FUNCTION_BLOCK ResetModulesVisitor IMPLEMENTS I_ModuleVisitor, I_TaskResult
VAR
	{attribute 'hide'}
	Resettable : I_Resettable;
	{attribute 'hide'}
	Result : I_TaskResult;
	{attribute 'hide'}
	_Busy : BOOL;
	{attribute 'hide'}
	_Error : BOOL;
	{attribute 'hide'}
	_ErrorId	: UDINT;
	ErrorModule : I_Module;
END_VAR

{attribute 'monitoring' := 'call'}
PROPERTY Busy : BOOL
GET
Busy := _Busy;
END_GET
END_PROPERTY

{attribute 'monitoring' := 'call'}
PROPERTY Error : BOOL
GET
Error := _Error;
END_GET
END_PROPERTY

{attribute 'monitoring' := 'call'}
PROPERTY ErrorId : UDINT
GET
ErrorID := _ErrorID;
END_GET
END_PROPERTY

METHOD Reset
VAR_INPUT
	Module : I_Module;
END_VAR
_Error	 := FALSE;
_ErrorId := 0;
_Busy	 := FALSE;
Module.Modules.Accept(THIS^);
END_METHOD

METHOD VisitModule
VAR_INPUT
	Module : I_Module;
END_VAR
IF __QUERYINTERFACE(Module, Resettable) THEN
	Resettable.Reset();
END_IF

IF __QUERYINTERFACE(Module, Result) THEN
	IF Result.Error THEN
		ErrorModule := Module;
		_Error		:= TRUE;
		_ErrorId	:= Result.ErrorId;
	END_IF

	IF Result.Busy THEN
		_Busy := TRUE;
	END_IF
END_IF
END_METHOD

END_FUNCTION_BLOCK

(* stored: Version 1.1.0.1, ProductVersion 3.1.4026.18
   POU ResetModulesVisitor: Id {8c953db4-d0e2-4d22-a0d1-e5952b5fa103}, SpecialFunc None
   Property Busy: Id {1ce68cf0-e1e6-4615-9e75-a858f8adc8a6}
   Get Get: Id {2e1e558c-deef-4a14-87e2-6f52372e3d1b}
   Property Error: Id {fb26592a-22e0-4cca-a7f9-d0d9b07ff04b}
   Get Get: Id {974bbad7-243b-49ae-9cad-bd592799f33f}
   Property ErrorId: Id {5350401d-0546-43aa-bf99-f04868e92255}
   Get Get: Id {a21dda1f-d5e4-4323-b539-6ec98f3738f6}
   Method Reset: Id {422a6468-493a-4978-a0b0-414f0b6d5a1b}
   Method VisitModule: Id {07ceb6be-b5c1-4353-9504-37404fa187e2} *)
